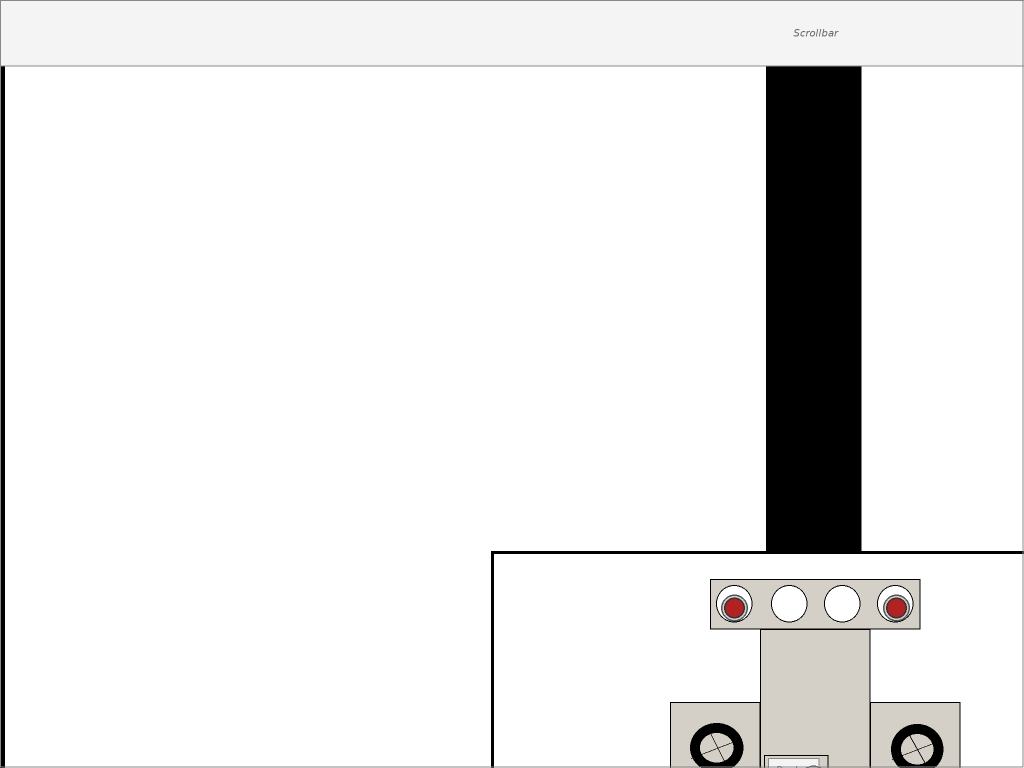
VISUALIZATION Visualization  // 1024x768
    Rectangle (0,0 1634x806)
    Rectangle (0,808 1581x618)
    Rectangle (766,-800 95x1565)
        p2858320360: LineAngle
    Rectangle (491,551 653x253)
    Group (670,579 290x221)
        Rectangle (0,123 90x90)
        Group (40,0 210x221)
            Rectangle (0,0 210x50)
            RoundedRectangle (50,50 110x171)
        Ellipse (207,6 36x37)
        Ellipse (46,6 36x37)
        Ellipse (154,6 36x37)
        Ellipse (101,6 36x37)
        Rectangle (200,123 90x90)
        Line (222,180) (271,161)
            p2858320360: POU_DT01_EnableDriveTrain.fbRightPower.Axis.NcToPlc.ActPos
        Line (21,179) (70,160)
            p2858320360: POU_DT01_EnableDriveTrain.fbLeftPower.Axis.NcToPlc.ActPos
        Ellipse (221,145 52x50)
        Ellipse (20,144 53x49)
        RoundedRectangle (94,176 64x42)
        RockerSwitch (98,179 51x37), tooltip "Turn off unit prior to Stopping runtime.", variable: SystemON, behaviour: TOGGLE, style: Switch-RockerSwitch-Gray
        Lamp1 (128,181 31x38), variable: SystemON, style: Lamp-Lamp1-Green
        Lamp1 (49,10 31x38), variable: LeftLimitExceeded, style: Lamp-Lamp1-Red
        Lamp1 (211,10 31x38), variable: RightLimitExceeded, style: Lamp-Lamp1-Red
        Line (258,189) (235,148)
            p2858320360: POU_DT01_EnableDriveTrain.fbRightPower.Axis.NcToPlc.ActPos
        Line (57,187) (37,147)
            p2858320360: POU_DT01_EnableDriveTrain.fbLeftPower.Axis.NcToPlc.ActPos
    Scrollbar (0,0 1632x66)
        p3598130195: -50
        p1057716461: LineAngle
    Meter180 (1235,461 250x250), value: LeftMotor.NcToPlc.ActVelo, style: Meter-Meter180-Gray, scale format: %.1f, scale 0..100
    BarDisplayImage (1207,652 300x50), value: RightMotor.NcToPlc.ActVelo, style: BarDisplayImage-Gray, scale format: %.1f, scale 0..100
END_VISUALIZATION

(* stored: Version 1.1.0.1, ProductVersion 3.1.4022.7
   Visu Visualization: Id {aa6a28f3-08bc-40db-a4d5-d24bf236b463} *)
